// TIA Portal V18 export
TYPE "RCS_SysCmd_V1"
   STRUCT
      Reset : Bool;   // Station Reset command
      ControlOff : Bool;   // PLC activate controll off command
      ChangeOver : Bool;   // Trigger Change Over command
      Record : Bool;
      TestLamp : Bool;
      BuzzerOn : Bool;
      StartRemember : Bool;
      Reserve : Bool;
      ClearFlags : Bool;   // Clear program Flags
      OnOffLine : Bool;
      OneCycle : Bool;   // Trigger one cycle running in Auto mode
      DryRun : Bool;   // Trigger dry cycle running in Auto mode
      Calibration : Bool;   // Special mode
   END_STRUCT;
END_TYPE
